TYPE Cnv_VTD_Control_DUT :
STRUCT
	Cnv_Level:	ARRAY[2..6] OF Cnv_Level_Control_DUT;
END_STRUCT
END_TYPE

(* stored: Version 1.1.0.1
   DUT Cnv_VTD_Control_DUT: Id {dae0fe20-e6e7-4986-8666-70dfb3c916d8} *)
